// Detect leaks and leak locations
FUNCTION_BLOCK FB_LeakMonitor
VAR_INPUT
	bLeakDetected : BOOL; // Whether a leak was detected
	bAmphosOn : BOOL; // Whether the Amphos is on
	bCarbideOn : BOOL; // Whether the Carbide is on
	nLocationResistance: UINT; // Used for calculating the location of the leak
END_VAR
VAR_IN_OUT CONSTANT
	stBoundaries : ST_LeakBoundaries; // Setpoints for calculating leak locations from location resistance
END_VAR
VAR_OUTPUT
	{attribute 'pytmc' := '
		pv: LOTAO_ERROR
		io: i
		field: OSV MAJOR
		field: ZSV NO_ALARM
		field: ZNAM OK
		field: ONAM ERROR
	'}
	bLeakOpticalTableAmphosOn : BOOL := FALSE; // Leak on the optical table with Amphos on
	{attribute 'pytmc' := '
		pv: LOTNL_ERROR
		io: i
		field: OSV MAJOR
		field: ZSV NO_ALARM
		field: ZNAM OK
		field: ONAM ERROR
	'}
	bLeakOpticalTableNoLaser : BOOL := FALSE; // Leak on the optical table with no laser on
	{attribute 'pytmc' := '
		pv: LOCO_ERROR
		io: i
		field: OSV MAJOR
		field: ZSV NO_ALARM
		field: ZNAM OK
		field: ONAM ERROR
	'}
	bLeakOpcpaCarbideOn : BOOL := FALSE; // Leak inside the OPCPA with Carbide on
	{attribute 'pytmc' := '
		pv: LUT_ERROR
		io: i
		field: OSV MAJOR
		field: ZSV NO_ALARM
		field: ZNAM OK
		field: ONAM ERROR
	'}
	bLeakUnderTable : BOOL := FALSE; // Leak under the table
	{attribute 'pytmc' := '
		pv: LIR_ERROR
		io: i
		field: OSV MAJOR
		field: ZSV NO_ALARM
		field: ZNAM OK
		field: ONAM ERROR
	'}
	bLeakInsideRacks : BOOL := FALSE; // Leak inside the racks
END_VAR
VAR
	{attribute 'pytmc' := '
		pv: LOC
		io: i
	'}
	eLeakLocation : E_LeakLocation := E_LeakLocation.NoLeak; // Location of the leak
END_VAR

// If there is a leak, detect the location of the leak and latch the error
IF bLeakDetected THEN
	IF stBoundaries.nLMin1 <= nLocationResistance AND nLocationResistance < stBoundaries.nLMax4 THEN
		IF bAmphosOn THEN
			eLeakLocation := E_LeakLocation.OpticalTable;
			bLeakOpticalTableAmphosOn := TRUE;
		ELSIF NOT bCarbideOn THEN
			eLeakLocation := E_LeakLocation.OpticalTable;
			bLeakOpticalTableNoLaser := TRUE;
		END_IF
	END_IF
	
	IF bCarbideOn AND stBoundaries.nLMin1 <= nLocationResistance AND nLocationResistance < stBoundaries.nLMax2 THEN
		eLeakLocation := E_LeakLocation.Opcpa;
		bLeakOpcpaCarbideOn := TRUE;
	END_IF
	
	IF stBoundaries.nLMin5 <= nLocationResistance AND nLocationResistance < stBoundaries.nLMax5 THEN
		eLeakLocation := E_LeakLocation.UnderTable;
		bLeakUnderTable := TRUE;
	END_IF
	
	IF stBoundaries.nLMin6 <= nLocationResistance AND nLocationResistance < stBoundaries.nLMax6 THEN
		eLeakLocation := E_LeakLocation.InsideRacks;
		bLeakInsideRacks := TRUE;
	END_IF
END_IF

// Reset latched errors
METHOD Reset
VAR_INPUT
END_VAR
eLeakLocation := E_LeakLocation.NoLeak;
bLeakOpticalTableAmphosOn := FALSE;
bLeakOpticalTableNoLaser := FALSE;
bLeakOpcpaCarbideOn := FALSE;
bLeakUnderTable := FALSE;
bLeakInsideRacks := FALSE;
END_METHOD

END_FUNCTION_BLOCK

(* stored: Version 1.1.0.1, ProductVersion 3.1.4020.14
   POU FB_LeakMonitor: Id {e43e7b93-d8f6-4d91-924b-e9e5b24db374}, SpecialFunc None
   Method Reset: Id {99e2e7d1-3dd4-4f42-8f02-0e9f34a50a59} *)
